// TwinCAT 3 PLC project M2K2
// ProgramVersion: 3.1.4022.7
// libraries:
//   LCLS General, * (SLAC)
//   lcls-twincat-motion, * (SLAC)
//   Tc2_MC2, * (Beckhoff Automation GmbH)
//   Tc2_Standard, * (Beckhoff Automation GmbH)
//   Tc2_System, * (Beckhoff Automation GmbH)
//   Tc3_Module, * (Beckhoff Automation GmbH)
// project tree:
//   / PlcTask.TcTTO
//   POUs/ FB_MotionStageStats.TcPOU, FB_PAT.TcPOU, Main.TcPOU
// real-time tasks:
//   TASK PlcTask: cycle T#10ms, priority 20, ADS port 350
// motion (NC):
//   TASK NC-Task 1 SAF: cycle T#2ms, priority 4, ADS port 501
//   TASK NC-Task 1 SVB: cycle T#10ms, priority 8, ADS port 511
//   AXIS M2K2 X (id 1)
//     OtherSettings: AllowMotionCmdToSlave=true
//     encoder EncType=29
//       EncPara: MaxCount=#xffffffff
//         Inc: RefSoftSyncMask=#x0000ffff
//     drive DrvType=24
//       Analog: ScaleFactorActTorque=0.1
//       TimeComp: TaskDelayCycles=1
//     controller CtrType=1
//       CtrPara: PriorControlFactor=1
//         Observer: BandWidth=20
//   AXIS M2K2 Y (id 2)
//     OtherSettings: AllowMotionCmdToSlave=true
//     encoder EncType=29
//       EncPara: MaxCount=#xffffffff
//         Inc: RefSoftSyncMask=#x0000ffff
//     drive DrvType=24
//       Analog: ScaleFactorActTorque=0.1
//       TimeComp: TaskDelayCycles=1
//     controller CtrType=1
//       CtrPara: PriorControlFactor=1
//         Observer: BandWidth=20
//   AXIS M2K2 rX (id 3)
//     OtherSettings: AllowMotionCmdToSlave=true
//     encoder EncType=29
//       EncPara: MaxCount=#xffffffff
//         Inc: RefSoftSyncMask=#x0000ffff
//     drive DrvType=24
//       Analog: ScaleFactorActTorque=0.1
//       TimeComp: TaskDelayCycles=1
//     controller CtrType=1
//       CtrPara: PriorControlFactor=1
//         Observer: BandWidth=20
// I/O:
//   DEVICE Device 1 (EtherCAT), AmsNetId 192.168.0.19.2.1
//     Term 1 (EK1100) [EK1100 EtherCAT Coupler (2A E-Bus)]
//       Term 2 (EL5042) [EL5042 2Ch. BiSS-C Encoder]
//       Term 3 (EL5042) [EL5042 2Ch. BiSS-C Encoder]
//       Term 4 (EL9221-5000) [EL9221-5000 Overcurrent protection 24V DC, 1Ch., max. 10A, adjustable]
//       M2K2 X
//       M2K2 Y
//       M2K2 rX
//       STO (EL1004) [EL1004 4Ch. Dig. Input 24V, 3ms]
//       Term 9 (EL9011) [EL9011 End Terminal]
// variable links:
//   NC-Task 1 SAF/Axes/M2K2 X <-> Device 1 (EtherCAT)/Term 1 (EK1100)/M2K2 X
//     Drive/Inputs/In/nState1 @bit 3 <-> STM Status/Status/Error
//     Drive/Inputs/In/nState1 @bit 5 <-> STM Status/Status/Moving negative
//     Drive/Inputs/In/nState1 @bit 4 <-> STM Status/Status/Moving positive
//     Drive/Inputs/In/nState1 @bit 1 <-> STM Status/Status/Ready
//     Drive/Inputs/In/nState1 <-> STM Status/Status/Ready to enable
//     Drive/Inputs/In/nState1 @bit 6 <-> STM Status/Status/Torque reduced
//     Drive/Inputs/In/nState1 @bit 2 <-> STM Status/Status/Warning
//     Drive/Inputs/In/nState2 @bit 3 <-> STM Status/Status/Digital input 1
//     Drive/Inputs/In/nState2 @bit 4 <-> STM Status/Status/Digital input 2
//     Drive/Inputs/In/nState2 @bit 5 <-> STM Status/Status/Sync error
//     Drive/Inputs/In/nState2 @bit 7 <-> STM Status/Status/TxPDO Toggle
//     Drive/Inputs/In/nState4 @bit 1 <-> WcState/InputToggle
//     Drive/Inputs/In/nState4 <-> WcState/WcState
//     Drive/Outputs/Out/nCtrl1 <-> STM Control/Control/Enable
//     Drive/Outputs/Out/nCtrl1 @bit 2 <-> STM Control/Control/Reduce torque
//     Drive/Outputs/Out/nCtrl1 @bit 1 <-> STM Control/Control/Reset
//     Drive/Outputs/Out/nDataOut2[0] <-> STM Velocity/Velocity
//   NC-Task 1 SAF/Axes/M2K2 X <-> Device 1 (EtherCAT)/Term 1 (EK1100)/Term 2 (EL5042)
//     Enc/Inputs/In/nComState @bit 1 <-> WcState/InputToggle
//     Enc/Inputs/In/nComState <-> WcState/WcState
//     Enc/Inputs/In/nDataIn1 <-> FB Inputs Channel 1/Position
//     Enc/Inputs/In/nState1 @bit 12 <-> FB Inputs Channel 1/Status/Diag
//     Enc/Inputs/In/nState1 @bit 1 <-> FB Inputs Channel 1/Status/Error
//     Enc/Inputs/In/nState1 @bit 14 <-> FB Inputs Channel 1/Status/Input cycle counter
//     Enc/Inputs/In/nState1 @bit 2 <-> FB Inputs Channel 1/Status/Ready
//     Enc/Inputs/In/nState1 @bit 13 <-> FB Inputs Channel 1/Status/TxPDO State
//     Enc/Inputs/In/nState1 <-> FB Inputs Channel 1/Status/Warning
//   NC-Task 1 SAF/Axes/M2K2 Y <-> Device 1 (EtherCAT)/Term 1 (EK1100)/M2K2 Y
//     Drive/Inputs/In/nState1 @bit 3 <-> STM Status/Status/Error
//     Drive/Inputs/In/nState1 @bit 5 <-> STM Status/Status/Moving negative
//     Drive/Inputs/In/nState1 @bit 4 <-> STM Status/Status/Moving positive
//     Drive/Inputs/In/nState1 @bit 1 <-> STM Status/Status/Ready
//     Drive/Inputs/In/nState1 <-> STM Status/Status/Ready to enable
//     Drive/Inputs/In/nState1 @bit 6 <-> STM Status/Status/Torque reduced
//     Drive/Inputs/In/nState1 @bit 2 <-> STM Status/Status/Warning
//     Drive/Inputs/In/nState2 @bit 3 <-> STM Status/Status/Digital input 1
//     Drive/Inputs/In/nState2 @bit 4 <-> STM Status/Status/Digital input 2
//     Drive/Inputs/In/nState2 @bit 5 <-> STM Status/Status/Sync error
//     Drive/Inputs/In/nState2 @bit 7 <-> STM Status/Status/TxPDO Toggle
//     Drive/Inputs/In/nState4 @bit 1 <-> WcState/InputToggle
//     Drive/Inputs/In/nState4 <-> WcState/WcState
//     Drive/Outputs/Out/nCtrl1 <-> STM Control/Control/Enable
//     Drive/Outputs/Out/nCtrl1 @bit 2 <-> STM Control/Control/Reduce torque
//     Drive/Outputs/Out/nCtrl1 @bit 1 <-> STM Control/Control/Reset
//     Drive/Outputs/Out/nDataOut2[0] <-> STM Velocity/Velocity
//   NC-Task 1 SAF/Axes/M2K2 Y <-> Device 1 (EtherCAT)/Term 1 (EK1100)/Term 2 (EL5042)
//     Enc/Inputs/In/nComState @bit 1 <-> WcState/InputToggle
//     Enc/Inputs/In/nComState <-> WcState/WcState
//     Enc/Inputs/In/nDataIn1 <-> FB Inputs Channel 2/Position
//     Enc/Inputs/In/nState1 @bit 12 <-> FB Inputs Channel 2/Status/Diag
//     Enc/Inputs/In/nState1 @bit 1 <-> FB Inputs Channel 2/Status/Error
//     Enc/Inputs/In/nState1 @bit 14 <-> FB Inputs Channel 2/Status/Input cycle counter
//     Enc/Inputs/In/nState1 @bit 2 <-> FB Inputs Channel 2/Status/Ready
//     Enc/Inputs/In/nState1 @bit 13 <-> FB Inputs Channel 2/Status/TxPDO State
//     Enc/Inputs/In/nState1 <-> FB Inputs Channel 2/Status/Warning
//   NC-Task 1 SAF/Axes/M2K2 rX <-> Device 1 (EtherCAT)/Term 1 (EK1100)/M2K2 rX
//     Drive/Inputs/In/nState1 @bit 3 <-> STM Status/Status/Error
//     Drive/Inputs/In/nState1 @bit 5 <-> STM Status/Status/Moving negative
//     Drive/Inputs/In/nState1 @bit 4 <-> STM Status/Status/Moving positive
//     Drive/Inputs/In/nState1 @bit 1 <-> STM Status/Status/Ready
//     Drive/Inputs/In/nState1 <-> STM Status/Status/Ready to enable
//     Drive/Inputs/In/nState1 @bit 6 <-> STM Status/Status/Torque reduced
//     Drive/Inputs/In/nState1 @bit 2 <-> STM Status/Status/Warning
//     Drive/Inputs/In/nState2 @bit 3 <-> STM Status/Status/Digital input 1
//     Drive/Inputs/In/nState2 @bit 4 <-> STM Status/Status/Digital input 2
//     Drive/Inputs/In/nState2 @bit 5 <-> STM Status/Status/Sync error
//     Drive/Inputs/In/nState2 @bit 7 <-> STM Status/Status/TxPDO Toggle
//     Drive/Inputs/In/nState4 @bit 1 <-> WcState/InputToggle
//     Drive/Inputs/In/nState4 <-> WcState/WcState
//     Drive/Outputs/Out/nCtrl1 <-> STM Control/Control/Enable
//     Drive/Outputs/Out/nCtrl1 @bit 2 <-> STM Control/Control/Reduce torque
//     Drive/Outputs/Out/nCtrl1 @bit 1 <-> STM Control/Control/Reset
//     Drive/Outputs/Out/nDataOut2[0] <-> STM Velocity/Velocity
//   NC-Task 1 SAF/Axes/M2K2 rX <-> Device 1 (EtherCAT)/Term 1 (EK1100)/Term 3 (EL5042)
//     Enc/Inputs/In/nComState @bit 1 <-> WcState/InputToggle
//     Enc/Inputs/In/nComState <-> WcState/WcState
//     Enc/Inputs/In/nDataIn1 <-> FB Inputs Channel 1/Position
//     Enc/Inputs/In/nState1 @bit 12 <-> FB Inputs Channel 1/Status/Diag
//     Enc/Inputs/In/nState1 @bit 1 <-> FB Inputs Channel 1/Status/Error
//     Enc/Inputs/In/nState1 @bit 14 <-> FB Inputs Channel 1/Status/Input cycle counter
//     Enc/Inputs/In/nState1 @bit 2 <-> FB Inputs Channel 1/Status/Ready
//     Enc/Inputs/In/nState1 @bit 13 <-> FB Inputs Channel 1/Status/TxPDO State
//     Enc/Inputs/In/nState1 <-> FB Inputs Channel 1/Status/Warning
//   M2K2/M2K2 Instance <-> Device 1 (EtherCAT)/Term 1 (EK1100)/M2K2 X
//     PlcTask Inputs/Main.M1.bLimitBackwardEnable <-> STM Status/Status/Digital input 2
//     PlcTask Inputs/Main.M1.bLimitForwardEnable <-> STM Status/Status/Digital input 1
//   M2K2/M2K2 Instance <-> Device 1 (EtherCAT)/Term 1 (EK1100)/M2K2 Y
//     PlcTask Inputs/Main.M2.bLimitBackwardEnable <-> STM Status/Status/Digital input 2
//     PlcTask Inputs/Main.M2.bLimitForwardEnable <-> STM Status/Status/Digital input 1
//   M2K2/M2K2 Instance <-> Device 1 (EtherCAT)/Term 1 (EK1100)/M2K2 rX
//     PlcTask Inputs/Main.M3.bLimitBackwardEnable <-> STM Status/Status/Digital input 2
//     PlcTask Inputs/Main.M3.bLimitForwardEnable <-> STM Status/Status/Digital input 1
//   M2K2/M2K2 Instance <-> Device 1 (EtherCAT)/Term 1 (EK1100)/STO (EL1004)
//     PlcTask Inputs/Main.bSTOEnable1 <-> Channel 1/Input
//     PlcTask Inputs/Main.bSTOEnable2 <-> Channel 2/Input
//   M2K2/M2K2 Instance <-> NC-Task 1 SAF/Axes/M2K2 X
//     PlcTask Inputs/Main.M1.Axis.NcToPlc <-> Outputs/ToPlc
//     PlcTask Outputs/Main.M1.Axis.PlcToNc <-> Inputs/FromPlc
//   M2K2/M2K2 Instance <-> NC-Task 1 SAF/Axes/M2K2 Y
//     PlcTask Inputs/Main.M2.Axis.NcToPlc <-> Outputs/ToPlc
//     PlcTask Outputs/Main.M2.Axis.PlcToNc <-> Inputs/FromPlc
//   M2K2/M2K2 Instance <-> NC-Task 1 SAF/Axes/M2K2 rX
//     PlcTask Inputs/Main.M3.Axis.NcToPlc <-> Outputs/ToPlc
//     PlcTask Outputs/Main.M3.Axis.PlcToNc <-> Inputs/FromPlc

CONFIGURATION M2K2
    RESOURCE PLC ON TwinCAT3
        TASK PlcTask(INTERVAL := T#10ms, PRIORITY := 20);
        PROGRAM Main WITH PlcTask : Main;
    END_RESOURCE
END_CONFIGURATION

// ---- POUs/Main.TcPOU
PROGRAM Main
VAR
	{attribute 'TcLinkTo' := '.bLimitForwardEnable:=TIIB[M2K2 X]^STM Status^Status^Digital input 1;
                              .bLimitBackwardEnable:=TIIB[M2K2 X]^STM Status^Status^Digital input 2'}
	M1 : DUT_MotionStage := (nEnableMode:=ENUM_StageEnableMode.DURING_MOTION);
	fbMotionStageM1 : FB_MotionStage;
	{attribute 'TcLinkTo' := '.bLimitForwardEnable:=TIIB[M2K2 Y]^STM Status^Status^Digital input 1;
                              .bLimitBackwardEnable:=TIIB[M2K2 Y]^STM Status^Status^Digital input 2'}
	M2 : DUT_MotionStage := (nEnableMode:=ENUM_StageEnableMode.DURING_MOTION);
	fbMotionStageM2 : FB_MotionStage;
	{attribute 'TcLinkTo' := '.bLimitForwardEnable:=TIIB[M2K2 rX]^STM Status^Status^Digital input 1;
                              .bLimitBackwardEnable:=TIIB[M2K2 rX]^STM Status^Status^Digital input 2'}
	M3 : DUT_MotionStage := (nEnableMode:=ENUM_StageEnableMode.DURING_MOTION);
	fbMotionStageM3 : FB_MotionStage;

	
	fbStepSizeTest_M2K2X : FB_MicroStepCountTest := (
		fStepSize := 0.00015625,
		nSteps := 1000,
		fMicroStep := 0.00015625,
		fVelocity := 1,
		tSettleTime := T#1S);
		
	fbStepSizeTest_M2K2Y : FB_MicroStepCountTest := (
		fStepSize := 0.0097656,
		nSteps := 1000,
		fMicroStep := 0.0097656,
		fVelocity := 0.5,
		tSettleTime := T#1S);
		
	fbStepSizeTest_M2K2rX : FB_MicroStepCountTest := (
		fStepSize := 0.0013021,
		nSteps := 1000,
		fMicroStep := 0.0013021,
		fVelocity := 10,
		tSettleTime := T#1S);
	
	fbM1Stats : FB_MotionStageStats;
	fbM2Stats : FB_MotionStageStats;
	fbM3Stats : FB_MotionStageStats;
	
	{attribute 'TcLinkTo' := 'TIID^Device 1 (EtherCAT)^Term 1 (EK1100)^STO (EL1004)^Channel 1^Input'}	
	bSTOEnable1 AT %I* : BOOL;
	{attribute 'TcLinkTo' := 'TIID^Device 1 (EtherCAT)^Term 1 (EK1100)^STO (EL1004)^Channel 2^Input'}
	bSTOEnable2 AT %I* : BOOL;
	
	END_VAR


M1.nEnableMode;
M2.nEnableMode;
M3.nEnableMode;

M1.bHardwareEnable := bSTOEnable1 AND bSTOEnable2;
M2.bHardwareEnable := bSTOEnable1 AND bSTOEnable2;
M3.bHardwareEnable := bSTOEnable1 AND bSTOEnable2;

fbMotionStageM1(stMotionStage:=M1);
fbMotionStageM2(stMotionStage:=M2);
fbMotionStageM3(stMotionStage:=M3);

fbM1Stats(Axis:=M1);
fbM2Stats(Axis:=M2);
fbM3Stats(Axis:=M3);

fbStepSizeTest_M2K2X(Axis:=M1.Axis);
fbStepSizeTest_M2K2Y(Axis:=M2.Axis);
fbStepSizeTest_M2K2rX(Axis:=M3.Axis);

END_PROGRAM

// ---- POUs/FB_MotionStageStats.TcPOU
FUNCTION_BLOCK FB_MotionStageStats EXTENDS FB_BasicStats
VAR_INPUT
	Axis : DUT_MotionStage;
END_VAR
VAR_OUTPUT
END_VAR
VAR
	aActPos : ARRAY [0..ARRAY_SIZE] OF LREAL;
	idx: UINT;
END_VAR
VAR CONSTANT
	ARRAY_SIZE : UINT := 500;
END_VAR


aActPos[idx] := Axis.Axis.NcToPlc.ActPos;

idx := (idx + 1) MOD ARRAY_SIZE;

SUPER^(aSignal:=aActPos, bAlwaysCalc:=NOT bReset);

END_FUNCTION_BLOCK

// ---- POUs/FB_PAT.TcPOU
FUNCTION_BLOCK FB_PAT
VAR_INPUT
    Velocity : LREAL;
END_VAR
VAR_OUTPUT
    FwLimPos : LREAL; // Positive limit position
    BwLimPos : LREAL; //
END_VAR
VAR_IN_OUT
    Stage : DUT_MotionStage;
END_VAR
VAR
    fbMicroStepCount : FB_MicroStepCountTest;

    fbMove: MC_Jog;
    tFwLim: F_TRIG;
    tBwLim: F_TRIG;
    Dir: INT;
END_VAR

// Relative move until limit, reverse and repeat, record positions, do math and spit out travel range

tFwLim(CLK:=Stage.bLimitForwardEnable);
tBwLim(CLK:=Stage.bLimitBackwardEnable);

WHILE Stage.bLimitBackwardEnable AND Stage.bLimitForwardEnable DO
    IF tFwLim.Q OR tBwLim.Q THEN
        IF (Dir = 1 AND tBwLim.Q) OR (Dir = -1 AND tFwLim.Q) THEN
            // Error, limits backwards
            EXIT;
        END_IF

        IF tFwLim.Q THEN
            FwLimPos := Stage.Axis.NcToPlc.ActPos;
        ELSIF tBwLim.Q THEN
            BwLimPos := Stage.Axis.NcToPlc.ActPos;
        END_IF


    END_IF



END_WHILE

// Discover minimum step size in one direction

// Attempt minimum step size in alternating direction

fbMove(Axis:=Stage.Axis, Velocity:=Velocity, Mode:=E_JogMode.MC_JOGMODE_CONTINOUS);

END_FUNCTION_BLOCK
